// Mitsubishi GX Works2 project: DanNhanTest   PLC: FX3G

PROGRAM MAIN
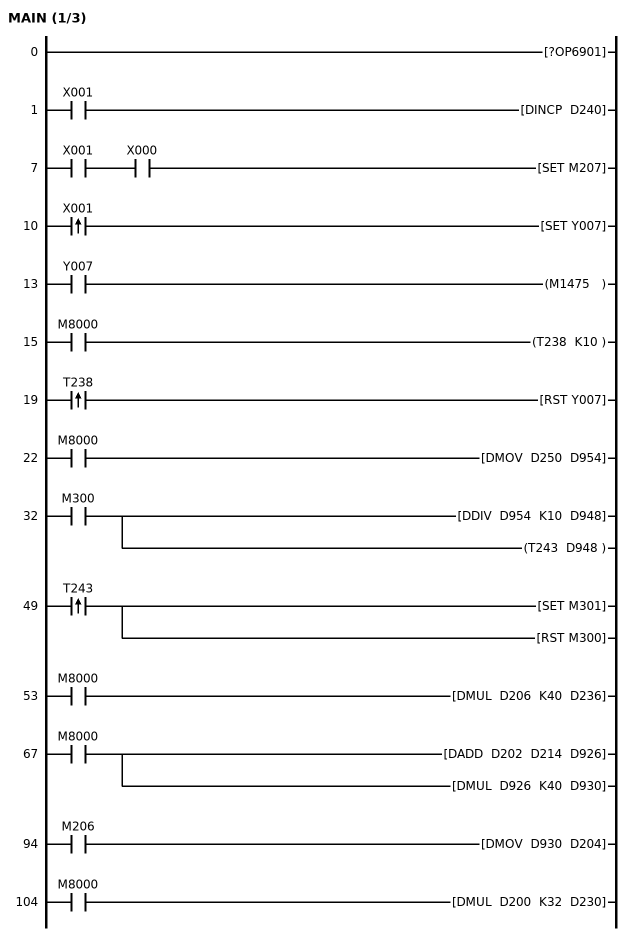
0     ?OP6901
1     LD      X001
      DINCP   D240
7     LD      X001
      AND     X000
      SET     M207
10    LDP     X001
      SET     Y007
13    LD      Y007
      OUT     M1475
15    LD      M8000
      OUT     T238 K10
19    LDP     T238
      RST     Y007
22    LD      M8000
      DMOV    D250 D954
32    LD      M300
      DDIV    D954 K10 D948
      OUT     T243 D948
49    LDP     T243
      SET     M301
      RST     M300
53    LD      M8000
      DMUL    D206 K40 D236
67    LD      M8000
      DADD    D202 D214 D926
      DMUL    D926 K40 D930
94    LD      M206
      DMOV    D930 D204
104   LD      M8000
      DMUL    D200 K32 D230
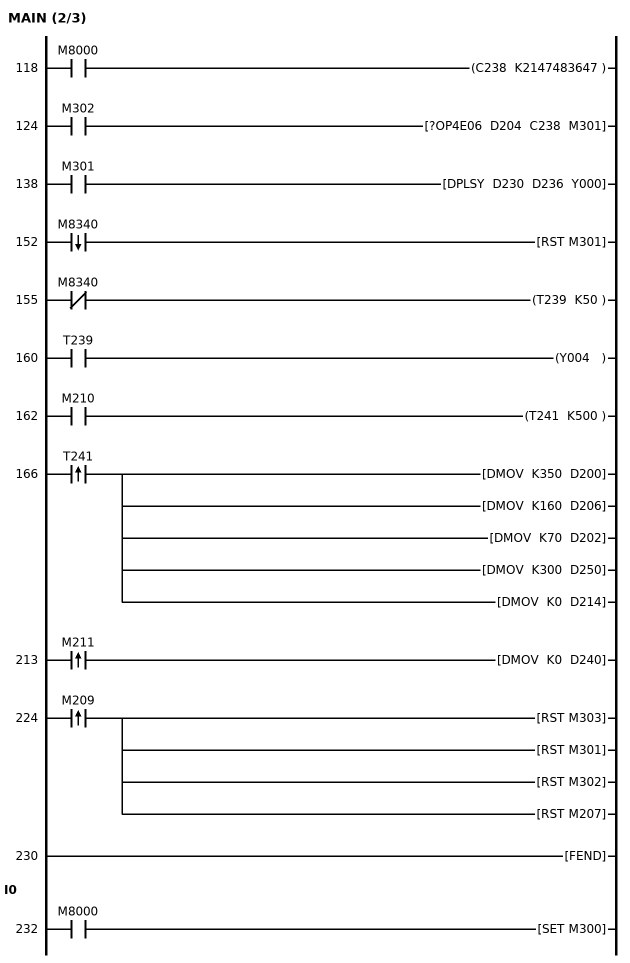
118   LD      M8000
      OUT     C238 K2147483647
124   LD      M302
      ?OP4E06 D204 C238 M301
138   LD      M301
      DPLSY   D230 D236 Y000
152   LDF     M8340
      RST     M301
155   LDI     M8340
      OUT     T239 K50
160   LD      T239
      OUT     Y004
162   LD      M210
      OUT     T241 K500
166   LDP     T241
      DMOV    K350 D200
      DMOV    K160 D206
      DMOV    K70 D202
      DMOV    K300 D250
      DMOV    K0 D214
213   LDP     M211
      DMOV    K0 D240
224   LDP     M209
      RST     M303
      RST     M301
      RST     M302
      RST     M207
230   FEND
      I0
232   LD      M8000
      SET     M300
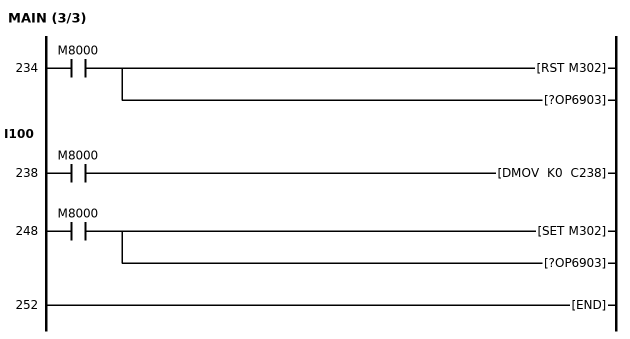
234   LD      M8000
      RST     M302
      ?OP6903
      I100
238   LD      M8000
      DMOV    K0 C238
248   LD      M8000
      SET     M302
      ?OP6903
252   END
END_PROGRAM
